// TIA Portal V19 export
FUNCTION_BLOCK "EXCHANGETRAY_EmStatusFeedBack"   // FB9, LAD
// stored: MemoryReserve 100, Namespace Unit3.EM1, SetENOAutomatically false
BEGIN

REGION Network 2 (SCL): stop：2

   IF ("Unit3.EM1.ControlNodes".sequence.status.currentStep>=100
       AND
       "Unit3.EM1.ControlNodes".sequence.status.currentStep<=199)
       OR
       ("Unit3.EM1.ControlNodes".sequence.status.currentStep>=300
       AND
       "Unit3.EM1.ControlNodes".sequence.status.currentStep<=499)
       OR
       ("Unit3.EM1.ControlNodes".sequence.status.currentStep>=600
       AND
       "Unit3.EM1.ControlNodes".sequence.status.currentStep<=799)
   THEN
       "Unit3.EmNodes".emStatus[Unit3_EM1].current:= 2;
   END_IF;
END_REGION

REGION Network 3 (SCL): execute：1
   IF
       ("Unit3.EM1.ControlNodes".sequence.status.currentStep>=203
       AND
       "Unit3.EM1.ControlNodes".sequence.status.currentStep<=299)





   THEN
       "Unit3.EmNodes".emStatus[Unit3_EM1].current := 1;
   END_IF;
END_REGION

REGION Network 4 (SCL): 暂停:40
   IF 
       "Unit3.EM1.ControlNodes".sequence.status.currentStep=201
       OR
       "Unit3.EM1.ControlNodes".sequence.status.currentStep=202
   THEN
       "Unit3.EmNodes".emStatus[Unit3_EM1].current := 40;
   END_IF;
END_REGION

REGION Network 5 (SCL): hold:20
   IF "Unit3.EmNodes".unitStatus.state.held

   THEN
       "Unit3.EmNodes".emStatus[Unit3_EM1].current :=20;
   END_IF;
END_REGION
END_FUNCTION_BLOCK
